TYPE ST_RepetitionArray :
STRUCT
	arrRepetition : ARRAY[1..10] OF DWORD;
END_STRUCT
END_TYPE

(* stored: Version 1.1.0.1, ProductVersion 3.1.4024.9
   DUT ST_RepetitionArray: Id {4238de6b-605c-4e86-823d-39c8da89ee6e} *)
